# EPICS substitutions: apps/jscalerApp/Db/wf/jscalers_wf_S1.substitutions
file "db/jscalers_wf_averages-1type-1sector.db" {
pattern { T S }
{ FADC 1 }
{ TRG 1 }
{ TDC 1 }
}
